FUNCTION_BLOCK FB_Controller EXTENDS FB_Object_Template_ST
VAR_INPUT
	//Discharger
	Tray_1 : BOOL; 
	Tray_2 : BOOL;
END_VAR
VAR_OUTPUT
	Fail : BOOL;
END_VAR
VAR
	Director   : FB_Director;
	Discharger : FB_Discharger_ST;
	Production : FB_F1Production_SFC;
	Panel      : FB_Panel;
	End: BOOL;
END_VAR

IC := Discharger.IC;
End := Production.Done;
Director(Emergency :=  Panel.Emergency,
		 Endbatch := Production.Done,
		 End := End,
		 Fail := Fail,
		 Go := Panel.Go,
		 Manual := Panel.Manual,
		 Reboot := Panel.Reboot,
		 Restore := IC,
		 Stop := Panel.Stop
		 );

Production(Execute := (Director.Mode=F1ProduccionNormal), 
			Ack :=Ack,
			SFCReset:=Reset,
			SFCPause :=Pause,
			IC:=IC,
			Discharger_Done:=Discharger.Done,
			);
			
		 
Panel (Mode := Director.Mode);

Discharger(Execute:=Production.Discharger_Execute,
			Ack:=Production.Discharger_Ack,
			Reset:=Reset,
			Pause:=Pause,
			Tray_1:=Tray_1,
			Tray_2:=Tray_2
			);

END_FUNCTION_BLOCK

(* stored: Version 1.1.0.1, ProductVersion 3.1.4024.6
   POU FB_Controller: Id {0de43ee4-da15-4690-902f-7120ea409570}, SpecialFunc None *)
